FUNCTION_BLOCK Skill_ROS2_Eyes EXTENDS FB_Template_ROS2Skill_V2
VAR_INPUT
	{attribute 'OPC.UA.DA.StructuredType':=1}
	{attribute 'OPC.UA.DA' := '1'}
	Specific    : ST_EyesSpecific;
END_VAR
VAR_OUTPUT
END_VAR
VAR
END_VAR

END_FUNCTION_BLOCK

(* stored: Version 1.1.0.1, ProductVersion 3.1.4026.18
   POU Skill_ROS2_Eyes: Id {db69cf7f-5a07-4e35-bdc2-21f16fa8d83c}, SpecialFunc None *)
